	  // "PACKMLV2022".Admin.DisabledStatesCfg["LPMLV2022_MODE_INVALID"]     := "InstLPMLV2022_UnitModeStateManager".configuration.DisabledStatesCfg["LPMLV2022_MODE_INVALID"];
	  "PACKMLV2022".Admin.DisabledStatesCfg["LPMLV2022_MODE_PRODUCTION"]  := "InstLPMLV2022_UnitModeStateManager".configuration.DisabledStatesCfg["LPMLV2022_MODE_PRODUCTION"];
	  "PACKMLV2022".Admin.DisabledStatesCfg["LPMLV2022_MODE_MAINTENANCE"] := "InstLPMLV2022_UnitModeStateManager".configuration.DisabledStatesCfg["LPMLV2022_MODE_MAINTENANCE"];
	  "PACKMLV2022".Admin.DisabledStatesCfg["LPMLV2022_MODE_MANUAL"]      := "InstLPMLV2022_UnitModeStateManager".configuration.DisabledStatesCfg["LPMLV2022_MODE_MANUAL"];
	  "PACKMLV2022".Admin.DisabledStatesCfg["LPMLV2022_MODE_USER_01"]     := "InstLPMLV2022_UnitModeStateManager".configuration.DisabledStatesCfg["LPMLV2022_MODE_USER_01"];
	  // "PACKMLV2022".Admin.DisabledStatesCfg["LPMLV2022_MODE_USER_02"]     := "InstLPMLV2022_UnitModeStateManager".configuration.DisabledStatesCfg["LPMLV2022_MODE_USER_02"];
	  
	  "PACKMLV2022".Admin.CurDisabledStates := "InstLPMLV2022_UnitModeStateManager".CurDisabledStates;
	  
	  "PACKMLV2022".Admin.EnabledModesCfg := "InstLPMLV2022_UnitModeStateManager".configuration.EnabledModesCfg;
	  
	  // "PACKMLV2022".Admin.ModeTransitionCfg["LPMLV2022_MODE_INVALID"]     := "InstLPMLV2022_UnitModeStateManager".configuration.ModeTransitionCfg["LPMLV2022_MODE_INVALID"];
	  "PACKMLV2022".Admin.ModeTransitionCfg["LPMLV2022_MODE_PRODUCTION"]  := "InstLPMLV2022_UnitModeStateManager".configuration.ModeTransitionCfg["LPMLV2022_MODE_PRODUCTION"];
	  "PACKMLV2022".Admin.ModeTransitionCfg["LPMLV2022_MODE_MAINTENANCE"] := "InstLPMLV2022_UnitModeStateManager".configuration.ModeTransitionCfg["LPMLV2022_MODE_MAINTENANCE"];
	  "PACKMLV2022".Admin.ModeTransitionCfg["LPMLV2022_MODE_MANUAL"]      := "InstLPMLV2022_UnitModeStateManager".configuration.ModeTransitionCfg["LPMLV2022_MODE_MANUAL"];
	  "PACKMLV2022".Admin.ModeTransitionCfg["LPMLV2022_MODE_USER_01"]     := "InstLPMLV2022_UnitModeStateManager".configuration.ModeTransitionCfg["LPMLV2022_MODE_USER_01"];
	  // "PACKMLV2022".Admin.ModeTransitionCfg["LPMLV2022_MODE_USER_02"]     := "InstLPMLV2022_UnitModeStateManager".configuration.ModeTransitionCfg["LPMLV2022_MODE_USER_02"];
	  
	  // PLCDateTime
	  #tempReturnValue := RD_LOC_T(#tempPLCDateTimeDTL);
	  
	  "PACKMLV2022".Admin.PLCDateTime.Year        := UINT_TO_INT(#tempPLCDateTimeDTL.YEAR);
	  "PACKMLV2022".Admin.PLCDateTime.Month       := #tempPLCDateTimeDTL.MONTH;
	  "PACKMLV2022".Admin.PLCDateTime.Day         := #tempPLCDateTimeDTL.DAY;
	  "PACKMLV2022".Admin.PLCDateTime.Hour        := #tempPLCDateTimeDTL.HOUR;
	  "PACKMLV2022".Admin.PLCDateTime.Minute      := #tempPLCDateTimeDTL.MINUTE;
	  "PACKMLV2022".Admin.PLCDateTime.Second      := #tempPLCDateTimeDTL.SECOND;
	  "PACKMLV2022".Admin.PLCDateTime.Millisecond := UDINT_TO_INT(#tempPLCDateTimeDTL.NANOSECOND / 1000000);
	  
	  "PACKMLV2022".Admin.PLCDateTimeDTL := #tempPLCDateTimeDTL;
	END_REGION
END_FUNCTION_BLOCK

FUNCTION_BLOCK "LPMLV2022_UnitModeStateManagerBool"
TITLE = LPMLV2022_UnitModeStateManagerBool
{ S7_Optimized_Access := 'TRUE' }
AUTHOR : APC_ERLF
FAMILY : OMAC
VERSION : 1.0
//Support: tech.team.motioncontrol@siemens.com
   VAR_INPUT 
      ProductionModeRequest { S7_HiddenAssignment := 'Show'} : Bool;   // Rising edge: Request change to unit mode Production
      MaintenanceModeRequest { S7_HiddenAssignment := 'Show'} : Bool;   // Rising edge: Request change to unit mode Maintenance
      ManualModeRequest { S7_HiddenAssignment := 'Show'} : Bool;   // Rising edge: Request change to unit mode Manual
      UserMode01Request { S7_HiddenAssignment := 'Show'} : Bool;   // Rising edge: Request change to user-defined unit mode 01
      UserMode02Request : Bool;   // Rising edge: Request change to user-defined unit mode 02
      UserMode03Request : Bool;   // Rising edge: Request change to user-defined unit mode 03
      UserMode04Request : Bool;   // Rising edge: Request change to user-defined unit mode 04
      UserMode05Request : Bool;   // Rising edge: Request change to user-defined unit mode 05
      ResetCmdRequest { S7_HiddenAssignment := 'Show'} : Bool;   // Rising edge: Request control command Reset
      StartCmdRequest { S7_HiddenAssignment := 'Show'} : Bool;   // Rising edge: Request control command Start
      StopCmdRequest { S7_HiddenAssignment := 'Show'} : Bool;   // Rising edge: Request control command Stop
      HoldCmdRequest { S7_HiddenAssignment := 'Show'} : Bool;   // Rising edge: Request control command Hold
      UnholdCmdRequest { S7_HiddenAssignment := 'Show'} : Bool;   // Rising edge: Request control command Unhold
      SuspendCmdRequest { S7_HiddenAssignment := 'Show'} : Bool;   // Rising edge: Request control command Suspend
      UnsuspendCmdRequest { S7_HiddenAssignment := 'Show'} : Bool;   // Rising edge: Request control command Unsuspend
      AbortCmdRequest { S7_HiddenAssignment := 'Show'} : Bool;   // Rising edge: Request control command Abort
      ClearCmdRequest { S7_HiddenAssignment := 'Show'} : Bool;   // Rising edge: Request control command Clear
      CompleteCmdRequest { S7_HiddenAssignment := 'Show'} : Bool;   // Rising edge: Request control command Complete
      SC : Bool;   // State change from FALSE to TRUE (rising edge) triggers state complete signal
      configuration : "LPMLV2022_typeConfiguration" := ((), [()], [16#0, 31(16#0000_0214)], (), ());   // FB configuration (is taken into account in first call after STOP/RUN)
   END_VAR

   VAR_OUTPUT 
      UnitModeCurrent { ExternalWritable := 'False'} : DInt := "LPMLV2022_MODE_INVALID";   // Current unit mode
      StateCurrent { ExternalWritable := 'False'} : DInt := "LPMLV2022_STATE_UNDEFINED";   // Current state
      ProductionModeActive { ExternalWritable := 'False'; S7_HiddenAssignment := 'Show'} : Bool;   // TRUE: Unit mode Production is currently active
      MaintenanceModeActive { ExternalWritable := 'False'; S7_HiddenAssignment := 'Show'} : Bool;   // TRUE: Unit mode Maintenance is currently active
      ManualModeActive { ExternalWritable := 'False'; S7_HiddenAssignment := 'Show'} : Bool;   // TRUE: Unit mode Manual is currently active
      UserMode01Active { ExternalWritable := 'False'; S7_HiddenAssignment := 'Show'} : Bool;   // TRUE: User-defined unit mode 01 is currently active
      UserMode02Active { ExternalWritable := 'False'} : Bool;   // TRUE: User-defined unit mode 02 is currently active
      UserMode03Active { ExternalWritable := 'False'} : Bool;   // TRUE: User-defined unit mode 03 is currently active
      UserMode04Active { ExternalWritable := 'False'} : Bool;   // TRUE: User-defined unit mode 04 is currently active
      UserMode05Active { ExternalWritable := 'False'} : Bool;   // TRUE: User-defined unit mode 05 is currently active
      ClearingStateActive { ExternalWritable := 'False'; S7_HiddenAssignment := 'Show'} : Bool;   // TRUE: State Clearing is currently active
      StoppedStateActive { ExternalWritable := 'False'; S7_HiddenAssignment := 'Show'} : Bool;   // TRUE: State Stopped is currently active
      StartingStateActive { ExternalWritable := 'False'; S7_HiddenAssignment := 'Show'} : Bool;   // TRUE: State Starting is currently active
      IdleStateActive { ExternalWritable := 'False'; S7_HiddenAssignment := 'Show'} : Bool;   // TRUE: State Idle is currently active
      SuspendedStateActive { ExternalWritable := 'False'; S7_HiddenAssignment := 'Show'} : Bool;   // TRUE: State Suspended is currently active
      ExecuteStateActive { ExternalWritable := 'False'; S7_HiddenAssignment := 'Show'} : Bool;   // TRUE: State Execute is currently active
      StoppingStateActive { ExternalWritable := 'False'; S7_HiddenAssignment := 'Show'} : Bool;   // TRUE: State Stopping is currently active
      AbortingStateActive { ExternalWritable := 'False'; S7_HiddenAssignment := 'Show'} : Bool;   // TRUE: State Aborting is currently active
      AbortedStateActive { ExternalWritable := 'False'; S7_HiddenAssignment := 'Show'} : Bool;   // TRUE: State Aborted is currently active
      HoldingStateActive { ExternalWritable := 'False'; S7_HiddenAssignment := 'Show'} : Bool;   // TRUE: State Holding is currently active
      HeldStateActive { ExternalWritable := 'False'; S7_HiddenAssignment := 'Show'} : Bool;   // TRUE: State Held is currently active
      UnholdingStateActive { ExternalWritable := 'False'; S7_HiddenAssignment := 'Show'} : Bool;   // TRUE: State Unholding is currently active
      SuspendingStateActive { ExternalWritable := 'False'; S7_HiddenAssignment := 'Show'} : Bool;   // TRUE: State Suspending is currently active
      UnsuspendingStateActive { ExternalWritable := 'False'; S7_HiddenAssignment := 'Show'} : Bool;   // TRUE: State Unsuspending is currently active
      ResettingStateActive { ExternalWritable := 'False'; S7_HiddenAssignment := 'Show'} : Bool;   // TRUE: State Resetting is currently active
      CompletingStateActive { ExternalWritable := 'False'; S7_HiddenAssignment := 'Show'} : Bool;   // TRUE: State Completing is currently active
      CompletedStateActive { ExternalWritable := 'False'; S7_HiddenAssignment := 'Show'} : Bool;   // TRUE: State Completed is currently active
      unitModeChangeNotAllowed { ExternalWritable := 'False'} : Bool;   // TRUE: Requested unit mode change is not allowed (output is reset with the next successful unit mode change or if all corresponding request inputs are set to FALSE)
      cntrlCmdNotAllowed { ExternalWritable := 'False'} : Bool;   // TRUE: Control command is not allowed (output is reset with the next successful control command or if all corresponding request inputs are set to FALSE)
   END_VAR

   VAR 
      instUnitModeStateManager { ExternalWritable := 'False'; S7_SetPoint := 'False'} : "LPMLV2022_UnitModeStateManager";   // Instance of LPMLV2022_UnitModeStateManager
      statFirstCycle { ExternalAccessible := 'False'; ExternalVisible := 'False'; ExternalWritable := 'False'} : Bool := TRUE;   // First cycle of run
      statUnitModeCurrentInternalOld { ExternalAccessible := 'False'; ExternalVisible := 'False'; ExternalWritable := 'False'} : DInt := "LPMLV2022_MODE_INVALID";   // For edge detection
      statStateInternalOld { ExternalAccessible := 'False'; ExternalVisible := 'False'; ExternalWritable := 'False'} : DInt := "LPMLV2022_STATE_UNDEFINED";   // For edge detection
      statBooleanInterfaceModeOld { ExternalAccessible := 'False'; ExternalVisible := 'False'; ExternalWritable := 'False'} : DWord;   // For edge detection
      statBooleanInterfaceCmdOld { ExternalAccessible := 'False'; ExternalVisible := 'False'; ExternalWritable := 'False'} : Word;   // For edge detection
   END_VAR

   VAR_TEMP 
      tempBooleanInterfaceMode : DWord;   // Status of boolean Mode inputs
      tempBooleanInterfaceCmd : Word;   // Status of boolean Cmd inputs except abort and stop
   END_VAR


BEGIN
	REGION HEADER
	  //================================================================================
	  // SIEMENS AG
	  // (c)Copyright 2023 All Rights Reserved
	  //--------------------------------------------------------------------------------
	  // Library: LPMLV2022 
	  // Tested with: S7-1211 with FW version V4.2, S7-1511-1 PN with FW version V2.6
	  // Engineering: TIA Portal V15.1
	  // Restrictions: -
	  // Requirements: S7-1200 FW 4.2 / S7-1500 FW 2.6
	  // Functionality: Machine and Unit States according to ANSI/ISA-TR88.00.02-2022
	  //                (if the default settings are active at 'holdCmdCfg' and 'completeCmdCfg')
	  // Support: tech.team.motioncontrol@siemens.com
	  // Note: Parameter comments are only available in language 'English (United States)'
	  //--------------------------------------------------------------------------------
	  // Change log table:
	  // Version  Date        Expert in charge  Changes applied
	  // 01.00.00 28.02.2023  KT                First released version
	  //================================================================================
	END_REGION
	
	IF #statFirstCycle THEN // Initialize values in first cycle
	  #instUnitModeStateManager.configuration := #configuration; // Copy configuration from input
	  #statFirstCycle := FALSE;
	
	ELSE // As from second cycle
	  //--------------------------------------------------------------------------------------------------
	  // Evaluation of input parameters
	  //--------------------------------------------------------------------------------------------------
	  #instUnitModeStateManager.UnitModeChangeRequest := TRUE; // Change request static TRUE
	
	  // Collect unit mode from boolean inputs
	  #tempBooleanInterfaceMode.%X1  := #ProductionModeRequest;
	  #tempBooleanInterfaceMode.%X2  := #MaintenanceModeRequest;
	  #tempBooleanInterfaceMode.%X3  := #ManualModeRequest;
	  #tempBooleanInterfaceMode.%X4  := #UserMode01Request;
	  #tempBooleanInterfaceMode.%X5  := #UserMode02Request;
	  #tempBooleanInterfaceMode.%X6  := #UserMode03Request;
	  #tempBooleanInterfaceMode.%X7  := #UserMode04Request;
	  #tempBooleanInterfaceMode.%X8  := #UserMode05Request;
	// #tempBooleanInterfaceMode.%X9  := #UserMode06Request;
	// #tempBooleanInterfaceMode.%X10 := #UserMode07Request;
	// #tempBooleanInterfaceMode.%X11 := #UserMode08Request;
	// #tempBooleanInterfaceMode.%X12 := #UserMode09Request;
	// #tempBooleanInterfaceMode.%X13 := #UserMode10Request;
	// #tempBooleanInterfaceMode.%X14 := #UserMode11Request;
	// #tempBooleanInterfaceMode.%X15 := #UserMode12Request;
	// #tempBooleanInterfaceMode.%X16 := #UserMode13Request;
	// #tempBooleanInterfaceMode.%X17 := #UserMode14Request;
	// #tempBooleanInterfaceMode.%X18 := #UserMode15Request;
	// #tempBooleanInterfaceMode.%X19 := #UserMode16Request;
	// #tempBooleanInterfaceMode.%X20 := #UserMode17Request;
	// #tempBooleanInterfaceMode.%X21 := #UserMode18Request;
	// #tempBooleanInterfaceMode.%X22 := #UserMode19Request;
	// #tempBooleanInterfaceMode.%X23 := #UserMode20Request;
	// #tempBooleanInterfaceMode.%X24 := #UserMode21Request;
	// #tempBooleanInterfaceMode.%X25 := #UserMode22Request;
	// #tempBooleanInterfaceMode.%X26 := #UserMode23Request;
	// #tempBooleanInterfaceMode.%X27 := #UserMode24Request;
	// #tempBooleanInterfaceMode.%X28 := #UserMode25Request;
	// #tempBooleanInterfaceMode.%X29 := #UserMode26Request;
	// #tempBooleanInterfaceMode.%X30 := #UserMode27Request;
	// #tempBooleanInterfaceMode.%X31 := #UserMode28Request;
	    
	  // Selection indicator: Rising edge at input, Priority (in case of multiple selection): Manual, Maintenance, User Mode 01..28, Production
	  IF #tempBooleanInterfaceMode.%X3 AND NOT #statBooleanInterfaceModeOld.%X3 THEN
	    #instUnitModeStateManager.UnitMode := "LPMLV2022_MODE_MANUAL";
	  ELSIF #tempBooleanInterfaceMode.%X2 AND NOT #statBooleanInterfaceModeOld.%X2 THEN
	    #instUnitModeStateManager.UnitMode := "LPMLV2022_MODE_MAINTENANCE";
	  ELSIF #tempBooleanInterfaceMode.%X4 AND NOT #statBooleanInterfaceModeOld.%X4 THEN
	    #instUnitModeStateManager.UnitMode := "LPMLV2022_MODE_USER_01";
	  ELSIF #tempBooleanInterfaceMode.%X5 AND NOT #statBooleanInterfaceModeOld.%X5 THEN
	    #instUnitModeStateManager.UnitMode := "LPMLV2022_MODE_USER_02";
	  ELSIF #tempBooleanInterfaceMode.%X6 AND NOT #statBooleanInterfaceModeOld.%X6 THEN
	    #instUnitModeStateManager.UnitMode := "LPMLV2022_MODE_USER_03";
	  ELSIF #tempBooleanInterfaceMode.%X7 AND NOT #statBooleanInterfaceModeOld.%X7 THEN
	    #instUnitModeStateManager.UnitMode := "LPMLV2022_MODE_USER_04";
	  ELSIF #tempBooleanInterfaceMode.%X8 AND NOT #statBooleanInterfaceModeOld.%X8 THEN
	    #instUnitModeStateManager.UnitMode := "LPMLV2022_MODE_USER_05";
	// ELSIF #tempBooleanInterfaceMode.%X9 AND NOT #statBooleanInterfaceModeOld.%X9 THEN
	//   #instUnitModeStateManager.UnitMode := "LPMLV2022_MODE_USER_06";
	// ELSIF #tempBooleanInterfaceMode.%X10 AND NOT #statBooleanInterfaceModeOld.%X10 THEN
	//   #instUnitModeStateManager.UnitMode := "LPMLV2022_MODE_USER_07";
	// ELSIF #tempBooleanInterfaceMode.%X11 AND NOT #statBooleanInterfaceModeOld.%X11 THEN
	//   #instUnitModeStateManager.UnitMode := "LPMLV2022_MODE_USER_08";
	// ELSIF #tempBooleanInterfaceMode.%X12 AND NOT #statBooleanInterfaceModeOld.%X12 THEN
	//   #instUnitModeStateManager.UnitMode := "LPMLV2022_MODE_USER_09";
	// ELSIF #tempBooleanInterfaceMode.%X13 AND NOT #statBooleanInterfaceModeOld.%X13 THEN
	//   #instUnitModeStateManager.UnitMode := "LPMLV2022_MODE_USER_10";
	// ELSIF #tempBooleanInterfaceMode.%X14 AND NOT #statBooleanInterfaceModeOld.%X14 THEN
	//   #instUnitModeStateManager.UnitMode := "LPMLV2022_MODE_USER_11";
	// ELSIF #tempBooleanInterfaceMode.%X15 AND NOT #statBooleanInterfaceModeOld.%X15 THEN
	//   #instUnitModeStateManager.UnitMode := "LPMLV2022_MODE_USER_12";
	// ELSIF #tempBooleanInterfaceMode.%X16 AND NOT #statBooleanInterfaceModeOld.%X16 THEN
	//   #instUnitModeStateManager.UnitMode := "LPMLV2022_MODE_USER_13";
	// ELSIF #tempBooleanInterfaceMode.%X17 AND NOT #statBooleanInterfaceModeOld.%X17 THEN
	//   #instUnitModeStateManager.UnitMode := "LPMLV2022_MODE_USER_14";
	// ELSIF #tempBooleanInterfaceMode.%X18 AND NOT #statBooleanInterfaceModeOld.%X18 THEN
	//   #instUnitModeStateManager.UnitMode := "LPMLV2022_MODE_USER_15";
	// ELSIF #tempBooleanInterfaceMode.%X19 AND NOT #statBooleanInterfaceModeOld.%X19 THEN
	//   #instUnitModeStateManager.UnitMode := "LPMLV2022_MODE_USER_16";
	// ELSIF #tempBooleanInterfaceMode.%X20 AND NOT #statBooleanInterfaceModeOld.%X20 THEN
	//   #instUnitModeStateManager.UnitMode := "LPMLV2022_MODE_USER_17";
	// ELSIF #tempBooleanInterfaceMode.%X21 AND NOT #statBooleanInterfaceModeOld.%X21 THEN
	//   #instUnitModeStateManager.UnitMode := "LPMLV2022_MODE_USER_18";
	// ELSIF #tempBooleanInterfaceMode.%X22 AND NOT #statBooleanInterfaceModeOld.%X22 THEN
	//   #instUnitModeStateManager.UnitMode := "LPMLV2022_MODE_USER_19";
	// ELSIF #tempBooleanInterfaceMode.%X23 AND NOT #statBooleanInterfaceModeOld.%X23 THEN
	//   #instUnitModeStateManager.UnitMode := "LPMLV2022_MODE_USER_20";
	// ELSIF #tempBooleanInterfaceMode.%X24 AND NOT #statBooleanInterfaceModeOld.%X24 THEN
	//   #instUnitModeStateManager.UnitMode := "LPMLV2022_MODE_USER_21";
	// ELSIF #tempBooleanInterfaceMode.%X25 AND NOT #statBooleanInterfaceModeOld.%X25 THEN
	//   #instUnitModeStateManager.UnitMode := "LPMLV2022_MODE_USER_22";
	// ELSIF #tempBooleanInterfaceMode.%X26 AND NOT #statBooleanInterfaceModeOld.%X26 THEN
	//   #instUnitModeStateManager.UnitMode := "LPMLV2022_MODE_USER_23";
	// ELSIF #tempBooleanInterfaceMode.%X27 AND NOT #statBooleanInterfaceModeOld.%X27 THEN
	//   #instUnitModeStateManager.UnitMode := "LPMLV2022_MODE_USER_24";
	// ELSIF #tempBooleanInterfaceMode.%X28 AND NOT #statBooleanInterfaceModeOld.%X28 THEN
	//   #instUnitModeStateManager.UnitMode := "LPMLV2022_MODE_USER_25";
	// ELSIF #tempBooleanInterfaceMode.%X29 AND NOT #statBooleanInterfaceModeOld.%X29 THEN
	//   #instUnitModeStateManager.UnitMode := "LPMLV2022_MODE_USER_26";
	// ELSIF #tempBooleanInterfaceMode.%X30 AND NOT #statBooleanInterfaceModeOld.%X30 THEN
	//   #instUnitModeStateManager.UnitMode := "LPMLV2022_MODE_USER_27";
	// ELSIF #tempBooleanInterfaceMode.%X31 AND NOT #statBooleanInterfaceModeOld.%X31 THEN
	//   #instUnitModeStateManager.UnitMode := "LPMLV2022_MODE_USER_28";
	  ELSIF #tempBooleanInterfaceMode.%X1 AND NOT #statBooleanInterfaceModeOld.%X1 THEN
	    #instUnitModeStateManager.UnitMode := "LPMLV2022_MODE_PRODUCTION";
	  ELSIF #tempBooleanInterfaceMode = 16#0000_0000 THEN // all corresponding boolean request inputs are FALSE
	    #instUnitModeStateManager.UnitMode := "LPMLV2022_MODE_INVALID";
	  END_IF;
	  
	  #statBooleanInterfaceModeOld := #tempBooleanInterfaceMode; // Save values for edge detection
	  
	  // State complete signal
	  #instUnitModeStateManager.SC := #SC;
	  
	  // Evaluate CntrlCmd in boolean interface; priority descending: abort, stop, other commands
	  #instUnitModeStateManager.CmdChangeRequest := TRUE; // Change request static TRUE
	  
	  #tempBooleanInterfaceCmd.%X1 := #ResetCmdRequest;
	  #tempBooleanInterfaceCmd.%X2 := #StartCmdRequest;
	  #tempBooleanInterfaceCmd.%X3 := #StopCmdRequest;
	  #tempBooleanInterfaceCmd.%X4 := #HoldCmdRequest;
	  #tempBooleanInterfaceCmd.%X5 := #UnholdCmdRequest;
	  #tempBooleanInterfaceCmd.%X6 := #SuspendCmdRequest;
	  #tempBooleanInterfaceCmd.%X7 := #UnsuspendCmdRequest;
	  #tempBooleanInterfaceCmd.%X8 := #AbortCmdRequest;
	  #tempBooleanInterfaceCmd.%X9 := #ClearCmdRequest;
	  #tempBooleanInterfaceCmd.%X10 := #CompleteCmdRequest;
	  
	  // Selection indicator: Rising edge at input, Priority (in case of multiple selection): abort, stop, complete, reset, start, hold, unhold, suspend, unsuspend, clear
	  IF #tempBooleanInterfaceCmd.%X8 AND NOT #statBooleanInterfaceCmdOld.%X8 THEN
	    #instUnitModeStateManager.CntrlCmd := "LPMLV2022_CMD_ABORT";
	  ELSIF #tempBooleanInterfaceCmd.%X3 AND NOT #statBooleanInterfaceCmdOld.%X3 THEN
	    #instUnitModeStateManager.CntrlCmd := "LPMLV2022_CMD_STOP";
	  ELSIF #tempBooleanInterfaceCmd.%X10 AND NOT #statBooleanInterfaceCmdOld.%X10 THEN
	    #instUnitModeStateManager.CntrlCmd := "LPMLV2022_CMD_COMPLETE";
	  ELSIF #tempBooleanInterfaceCmd.%X1 AND NOT #statBooleanInterfaceCmdOld.%X1 THEN
	    #instUnitModeStateManager.CntrlCmd := "LPMLV2022_CMD_RESET";
	  ELSIF #tempBooleanInterfaceCmd.%X2 AND NOT #statBooleanInterfaceCmdOld.%X2 THEN
	    #instUnitModeStateManager.CntrlCmd := "LPMLV2022_CMD_START";
	  ELSIF #tempBooleanInterfaceCmd.%X4 AND NOT #statBooleanInterfaceCmdOld.%X4 THEN
	    #instUnitModeStateManager.CntrlCmd := "LPMLV2022_CMD_HOLD";
	  ELSIF #tempBooleanInterfaceCmd.%X5 AND NOT #statBooleanInterfaceCmdOld.%X5 THEN
	    #instUnitModeStateManager.CntrlCmd := "LPMLV2022_CMD_UNHOLD";
	  ELSIF #tempBooleanInterfaceCmd.%X6 AND NOT #statBooleanInterfaceCmdOld.%X6 THEN
	    #instUnitModeStateManager.CntrlCmd := "LPMLV2022_CMD_SUSPEND";
	  ELSIF #tempBooleanInterfaceCmd.%X7 AND NOT #statBooleanInterfaceCmdOld.%X7 THEN
	    #instUnitModeStateManager.CntrlCmd := "LPMLV2022_CMD_UNSUSPEND";
	  ELSIF #tempBooleanInterfaceCmd.%X9 AND NOT #statBooleanInterfaceCmdOld.%X9 THEN
	    #instUnitModeStateManager.CntrlCmd := "LPMLV2022_CMD_CLEAR";
	  ELSIF #tempBooleanInterfaceCmd = 16#0000_0000 THEN // all corresponding boolean request inputs are FALSE
	    #instUnitModeStateManager.CntrlCmd := "LPMLV2022_CMD_UNDEFINED";
	  END_IF;
	  
	  #statBooleanInterfaceCmdOld := #tempBooleanInterfaceCmd; // Save values for edge detection
	END_IF;
	
	//--------------------------------------------------------------------------------------------------
	// Call unit mode state manager
	//--------------------------------------------------------------------------------------------------
	#instUnitModeStateManager();
	
	//--------------------------------------------------------------------------------------------------
	// Write outputs including boolean interface outputs 
	//--------------------------------------------------------------------------------------------------
	#UnitModeCurrent := #instUnitModeStateManager.UnitModeCurrent;
	#StateCurrent    := #instUnitModeStateManager.StateCurrent;
	
	IF #instUnitModeStateManager.UnitModeCurrent <> #statUnitModeCurrentInternalOld THEN // Check if new unit mode is selected
	  #ProductionModeActive := FALSE;
	  #MaintenanceModeActive := FALSE;
	  #ManualModeActive := FALSE;
	  #UserMode01Active := FALSE;
	  #UserMode02Active := FALSE;
	  #UserMode03Active := FALSE;
	  #UserMode04Active := FALSE;
	  #UserMode05Active := FALSE;
	  // #UserMode06Active := FALSE;
	  // #UserMode07Active := FALSE;
	  // #UserMode08Active := FALSE;
	  // #UserMode09Active := FALSE;
	  // #UserMode10Active := FALSE;
	  // #UserMode11Active := FALSE;
	  // #UserMode12Active := FALSE;
	  // #UserMode13Active := FALSE;
	  // #UserMode14Active := FALSE;
	  // #UserMode15Active := FALSE;
	  // #UserMode16Active := FALSE;
	  // #UserMode17Active := FALSE;
	  // #UserMode18Active := FALSE;
	  // #UserMode19Active := FALSE;
	  // #UserMode20Active := FALSE;
	  // #UserMode21Active := FALSE;
	  // #UserMode22Active := FALSE;
	  // #UserMode23Active := FALSE;
	  // #UserMode24Active := FALSE;
	  // #UserMode25Active := FALSE;
	  // #UserMode26Active := FALSE;
	  // #UserMode27Active := FALSE;
	  // #UserMode28Active := FALSE;
	  
	  CASE #instUnitModeStateManager.UnitModeCurrent OF // Set new bit for current unit mode
	    "LPMLV2022_MODE_PRODUCTION":
	      #ProductionModeActive := TRUE;
	    "LPMLV2022_MODE_MAINTENANCE":
	      #MaintenanceModeActive := TRUE;
	    "LPMLV2022_MODE_MANUAL":
	      #ManualModeActive := TRUE;
	    "LPMLV2022_MODE_USER_01":
	      #UserMode01Active := TRUE;
	    "LPMLV2022_MODE_USER_02":
	      #UserMode02Active := TRUE;
	    "LPMLV2022_MODE_USER_03":
	      #UserMode03Active := TRUE;
	    "LPMLV2022_MODE_USER_04":
	      #UserMode04Active := TRUE;
	    "LPMLV2022_MODE_USER_05":
	      #UserMode05Active := TRUE;
	    // "LPMLV2022_MODE_USER_06":
	    //   #UserMode06Active := TRUE;
	    // "LPMLV2022_MODE_USER_07":
	    //   #UserMode07Active := TRUE;
	    // "LPMLV2022_MODE_USER_08":
	    //   #UserMode08Active := TRUE;
	    // "LPMLV2022_MODE_USER_09":
	    //   #UserMode09Active := TRUE;
	    // "LPMLV2022_MODE_USER_10":
	    //   #UserMode10Active := TRUE;
	    // "LPMLV2022_MODE_USER_11":
	    //   #UserMode11Active := TRUE;
	    // "LPMLV2022_MODE_USER_12":
	    //   #UserMode12Active := TRUE;
	    // "LPMLV2022_MODE_USER_13":
	    //   #UserMode13Active := TRUE;
	    // "LPMLV2022_MODE_USER_14":
	    //   #UserMode14Active := TRUE;
	    // "LPMLV2022_MODE_USER_15":
	    //   #UserMode15Active := TRUE;
	    // "LPMLV2022_MODE_USER_16":
	    //   #UserMode16Active := TRUE;
	    // "LPMLV2022_MODE_USER_17":
	    //   #UserMode17Active := TRUE;
	    // "LPMLV2022_MODE_USER_18":
	    //   #UserMode18Active := TRUE;
	    // "LPMLV2022_MODE_USER_19":
	    //   #UserMode19Active := TRUE;
	    // "LPMLV2022_MODE_USER_2"0:
	    //   #UserMode20Active := TRUE;
	    // "LPMLV2022_MODE_USER_21":
	    //   #UserMode21Active := TRUE;
	    // "LPMLV2022_MODE_USER_22":
	    //   #UserMode22Active := TRUE;
	    // "LPMLV2022_MODE_USER_23":
	    //   #UserMode23Active := TRUE;
	    // "LPMLV2022_MODE_USER_24":
	    //   #UserMode24Active := TRUE;
	    // "LPMLV2022_MODE_USER_25":
	    //   #UserMode25Active := TRUE;
	    // "LPMLV2022_MODE_USER_26":
	    //   #UserMode26Active := TRUE;
	    // "LPMLV2022_MODE_USER_27":
	    //   #UserMode27Active := TRUE;
	    // "LPMLV2022_MODE_USER_28":
	    //   #UserMode28Active := TRUE;
	    ELSE
	      ; // No bit is set
	  END_CASE;
	  
	  #statUnitModeCurrentInternalOld := #instUnitModeStateManager.UnitModeCurrent;
	END_IF;
	
	IF #instUnitModeStateManager.StateCurrent <> #statStateInternalOld THEN // Check if new state is selected 
	  // Set states of boolean interface outputs
	  // Delete old state
	  #ClearingStateActive := FALSE;
	  #StoppedStateActive := FALSE;
	  #StartingStateActive := FALSE;
	  #IdleStateActive := FALSE;
	  #SuspendedStateActive := FALSE;
	  #ExecuteStateActive := FALSE;
	  #StoppingStateActive := FALSE;
	  #AbortingStateActive := FALSE;
	  #AbortedStateActive := FALSE;
	  #HoldingStateActive := FALSE;
	  #HeldStateActive := FALSE;
	  #UnholdingStateActive := FALSE;
	  #SuspendingStateActive := FALSE;
	  #UnsuspendingStateActive := FALSE;
	  #ResettingStateActive := FALSE;
	  #CompletingStateActive := FALSE;
	  #CompletedStateActive := FALSE;
	  
	  // Set new state
	  CASE #instUnitModeStateManager.StateCurrent OF
	    "LPMLV2022_STATE_CLEARING":
	      #ClearingStateActive := TRUE;
	    "LPMLV2022_STATE_STOPPED":
	      #StoppedStateActive := TRUE;
	    "LPMLV2022_STATE_STARTING":
	      #StartingStateActive := TRUE;
	    "LPMLV2022_STATE_IDLE":
	      #IdleStateActive := TRUE;
	    "LPMLV2022_STATE_SUSPENDED":
	      #SuspendedStateActive := TRUE;
	    "LPMLV2022_STATE_EXECUTE":
	      #ExecuteStateActive := TRUE;
	    "LPMLV2022_STATE_STOPPING":
	      #StoppingStateActive := TRUE;
	    "LPMLV2022_STATE_ABORTING":
	      #AbortingStateActive := TRUE;
	    "LPMLV2022_STATE_ABORTED":
	      #AbortedStateActive := TRUE;
	    "LPMLV2022_STATE_HOLDING":
	      #HoldingStateActive := TRUE;
	    "LPMLV2022_STATE_HELD":
	      #HeldStateActive := TRUE;
	    "LPMLV2022_STATE_UNHOLDING":
	      #UnholdingStateActive := TRUE;
	    "LPMLV2022_STATE_SUSPENDING":
	      #SuspendingStateActive := TRUE;
	    "LPMLV2022_STATE_UNSUSPENDING":
	      #UnsuspendingStateActive := TRUE;
	    "LPMLV2022_STATE_RESETTING":
	      #ResettingStateActive := TRUE;
	    "LPMLV2022_STATE_COMPLETING":
	      #CompletingStateActive := TRUE;
	    "LPMLV2022_STATE_COMPLETED":
	      #CompletedStateActive := TRUE;
	    ELSE
	      ;
	  END_CASE; // End: Set new state
	  
	  #statStateInternalOld := #instUnitModeStateManager.StateCurrent;
	END_IF;// End: Write boolean interface outputs
	
	#unitModeChangeNotAllowed := #instUnitModeStateManager.unitModeChangeNotAllowed;
	#cntrlCmdNotAllowed       := #instUnitModeStateManager.cntrlCmdNotAllowed;
END_FUNCTION_BLOCK

FUNCTION "LPMLV2022_ConfigureCompleteCmdCfg" : Void
TITLE = LPMLV2022_ConfigureCompleteCmdCfg
{ S7_Optimized_Access := 'TRUE' }
AUTHOR : APC_ERLF
FAMILY : OMAC
VERSION : 1.0
//Support: tech.team.motioncontrol@siemens.com
   VAR_INPUT 
      Suspended : Bool;   // TRUE: The Complete control command is taken into account in state Suspended
      Execute : Bool;   // TRUE: The Complete control command is taken into account in state Execute
      Held : Bool;   // TRUE: The Complete control command is taken into account in state Held
   END_VAR

   VAR_OUTPUT 
      completeCmdCfg : DWord;   // Complete control command configuration for all unit modes (one config. for all modes). Bit locations within the DWORD value represent State numbers
   END_VAR


BEGIN
	REGION HEADER
	  //================================================================================
	  // SIEMENS AG
	  // (c)Copyright 2023 All Rights Reserved
	  //--------------------------------------------------------------------------------
	  // Library: LPMLV2022
	  // Tested with: S7-1211 with FW version V4.2, S7-1511-1 PN with FW version V2.6
	  // Engineering: TIA Portal V15.1
	  // Restrictions: -
	  // Requirements: S7-1200 FW 4.2 / S7-1500 FW 2.6
	  // Functionality: The function generates a DWord value which represents
	  //                the state configuration for all unit modes.
	  //                
	  //                Note: All inputs must be set to comply with ANSI/ISA-TR88.00.02-2022
	  //
	  // Support: tech.team.motioncontrol@siemens.com
	  // Note: Parameter comments are only available in language 'English (United States)'
	  //--------------------------------------------------------------------------------
	  // Change log table:
	  // Version  Date        Expert in charge  Changes applied
	  // 01.00.00 28.02.2023  KT                First released version
	  //================================================================================
	END_REGION
	
	// Initialize states configuration
	#completeCmdCfg := 16#0000_0000;
	
	// Set states configuration
	#completeCmdCfg.%X5  := #Suspended;
	#completeCmdCfg.%X6  := #Execute;
	#completeCmdCfg.%X11 := #Held;
END_FUNCTION

FUNCTION "LPMLV2022_ConfigureHoldCmdCfg" : Void
TITLE = LPMLV2022_ConfigureHoldCmdCfg
{ S7_Optimized_Access := 'TRUE' }
AUTHOR : APC_ERLF
FAMILY : OMAC
VERSION : 1.0
//Support: tech.team.motioncontrol@siemens.com
   VAR_INPUT 
      Starting : Bool;   // TRUE: The Hold control command is taken into account in state Starting
      Idle : Bool;   // TRUE: The Hold control command is taken into account in state Idle
      Suspended : Bool;   // TRUE: The Hold control command is taken into account in state Suspended
      Execute : Bool;   // TRUE: The Hold control command is taken into account in state Execute
      Unholding : Bool;   // TRUE: The Hold control command is taken into account in state Unholding
      Suspending : Bool;   // TRUE: The Hold control command is taken into account in state Suspending
      Unsuspending : Bool;   // TRUE: The Hold control command is taken into account in state Unsuspending
      Completing : Bool;   // TRUE: The Hold control command is taken into account in state Completing
      Completed : Bool;   // TRUE: The Hold control command is taken into account in state Completed
   END_VAR

   VAR_OUTPUT 
      holdCmdCfg : DWord;   // Hold control command configuration for all unit modes (one config. for all modes). Bit locations within the DWORD value represent State numbers
   END_VAR


BEGIN
	REGION HEADER
	  //================================================================================
	  // SIEMENS AG
	  // (c)Copyright 2023 All Rights Reserved
	  //--------------------------------------------------------------------------------
	  // Library: LPMLV2022
	  // Tested with: S7-1211 with FW version V4.2, S7-1511-1 PN with FW version V2.6
	  // Engineering: TIA Portal V15.1
	  // Restrictions: -
	  // Requirements: S7-1200 FW 4.2 / S7-1500 FW 2.6
	  // Functionality: The function generates a DWord value which represents
	  //                the state configuration for all unit modes.
	  //                
	  //                Note: Only the inputs 'Suspended' and 'Execute' must be set
	  //                      to comply with ANSI/ISA-TR88.00.02-2022
	  //                      
	  // Support: tech.team.motioncontrol@siemens.com
	  // Note: Parameter comments are only available in language 'English (United States)'
	  //--------------------------------------------------------------------------------
	  // Change log table:
	  // Version  Date        Expert in charge  Changes applied
	  // 01.00.00 28.02.2023  KT                First released version
	  //================================================================================
	END_REGION
	
	// Initialize states configuration
	#holdCmdCfg := 16#0000_0000;
	
	// Set states configuration
	#holdCmdCfg.%X3  := #Starting;
	#holdCmdCfg.%X4  := #Idle;
	#holdCmdCfg.%X5  := #Suspended;
	#holdCmdCfg.%X6  := #Execute;
	#holdCmdCfg.%X12 := #Unholding;
	#holdCmdCfg.%X13 := #Suspending;
	#holdCmdCfg.%X14 := #Unsuspending;
	#holdCmdCfg.%X16 := #Completing;
	#holdCmdCfg.%X17 := #Completed;
END_FUNCTION

FUNCTION "LPMLV2022_ConfigureModeTransitionCfg" : Void
TITLE = LPMLV2022_ConfigureModeTransitionCfg
{ S7_Optimized_Access := 'TRUE' }
AUTHOR : APC_ERLF
FAMILY : OMAC
VERSION : 1.0
//Support: tech.team.motioncontrol@siemens.com
   VAR_INPUT 
      Clearing : Bool;   // TRUE: Allow a mode transition to/from state Clearing
      Stopped : Bool;   // TRUE: Allow a mode transition to/from state Stopped
      Starting : Bool;   // TRUE: Allow a mode transition to/from state Starting
      Idle : Bool;   // TRUE: Allow a mode transition to/from state Idle
      Suspended : Bool;   // TRUE: Allow a mode transition to/from state Suspended
      Execute : Bool;   // TRUE: Allow a mode transition to/from state Execute
      Stopping : Bool;   // TRUE: Allow a mode transition to/from state Stopping
      Aborting : Bool;   // TRUE: Allow a mode transition to/from state Aborting
      Aborted : Bool;   // TRUE: Allow a mode transition to/from state Aborted
      Holding : Bool;   // TRUE: Allow a mode transition to/from state Holding
      Held : Bool;   // TRUE: Allow a mode transition to/from state Held
      Unholding : Bool;   // TRUE: Allow a mode transition to/from state Unholding
      Suspending : Bool;   // TRUE: Allow a mode transition to/from state Suspending
      Unsuspending : Bool;   // TRUE: Allow a mode transition to/from state Unsuspending
      Resetting : Bool;   // TRUE: Allow a mode transition to/from state Resetting
      Completing : Bool;   // TRUE: Allow a mode transition to/from state Completing
      Completed : Bool;   // TRUE: Allow a mode transition to/from state Completed
   END_VAR

   VAR_OUTPUT 
      ModeTransitionCfg : DWord;   // Mode Transition Configuration for one unit mode. Bit locations within the DWORD value represent State numbers
   END_VAR


BEGIN
	REGION HEADER
	  //================================================================================
	  // SIEMENS AG
	  // (c)Copyright 2023 All Rights Reserved
	  //--------------------------------------------------------------------------------
	  // Library: LPMLV2022
	  // Tested with: S7-1211 with FW version V4.2, S7-1511-1 PN with FW version V2.6
	  // Engineering: TIA Portal V15.1
	  // Restrictions: -
	  // Requirements: S7-1200 FW 4.2 / S7-1500 FW 2.6
	  // Functionality: The function generates a DWord value which represents
	  //                the state configuration for one unit mode.
	  // Support: tech.team.motioncontrol@siemens.com
	  // Note: Parameter comments are only available in language 'English (United States)'
	  //--------------------------------------------------------------------------------
	  // Change log table:
	  // Version  Date        Expert in charge  Changes applied
	  // 01.00.00 28.02.2023  KT                First released version
	  //================================================================================
	END_REGION
	
	// Initialize states configuration
	#ModeTransitionCfg := 16#0000_0000;
	
	// Set states configuration
	#ModeTransitionCfg.%X1  := #Clearing;
	#ModeTransitionCfg.%X2  := #Stopped;
	#ModeTransitionCfg.%X3  := #Starting;
	#ModeTransitionCfg.%X4  := #Idle;
	#ModeTransitionCfg.%X5  := #Suspended;
	#ModeTransitionCfg.%X6  := #Execute;
	#ModeTransitionCfg.%X7  := #Stopping;
	#ModeTransitionCfg.%X8  := #Aborting;
	#ModeTransitionCfg.%X9  := #Aborted;
	#ModeTransitionCfg.%X10 := #Holding;
	#ModeTransitionCfg.%X11 := #Held;
	#ModeTransitionCfg.%X12 := #Unholding;
	#ModeTransitionCfg.%X13 := #Suspending;
	#ModeTransitionCfg.%X14 := #Unsuspending;
	#ModeTransitionCfg.%X15 := #Resetting;
	#ModeTransitionCfg.%X16 := #Completing;
	#ModeTransitionCfg.%X17 := #Completed;
END_FUNCTION

FUNCTION_BLOCK "LPMLV2022_Stacklight"
TITLE = LPMLV2022_Stacklight
{ S7_Optimized_Access := 'TRUE' }
AUTHOR : APC_ERLF
FAMILY : OMAC
VERSION : 1.0
//Support: tech.team.motioncontrol@siemens.com
   VAR_INPUT 
      StateCurrent : DInt := "LPMLV2022_STATE_UNDEFINED";   // Current state
      starvedUpstream : Bool;   // TRUE: upstream system is not able to supply products
      blockedDownstream : Bool;   // TRUE: downstream system is not able to accept products
      materialLow : Bool;   // TRUE: low material
      materialExhausted : Bool;   // TRUE: material exhausted
   END_VAR

   VAR_OUTPUT 
      Stacklight { ExternalWritable := 'False'} : DWord;   // Indicator for the current stacklight status -> PackTags
      redSolid { ExternalWritable := 'False'} : Bool;   // Status of stacklight bit 0
      redFlashing { ExternalWritable := 'False'} : Bool;   // Status of stacklight bit 1
      amberSolid { ExternalWritable := 'False'} : Bool;   // Status of stacklight bit 2
      amberFlashing { ExternalWritable := 'False'} : Bool;   // Status of stacklight bit 3
      blueSolid { ExternalWritable := 'False'} : Bool;   // Status of stacklight bit 4
      blueFlashing { ExternalWritable := 'False'} : Bool;   // Status of stacklight bit 5
      greenSolid { ExternalWritable := 'False'} : Bool;   // Status of stacklight bit 6
      greenFlashing { ExternalWritable := 'False'} : Bool;   // Status of stacklight bit 7
      hornFlashing { ExternalWritable := 'False'} : Bool;   // Status of stacklight bit 9
   END_VAR

   VAR_TEMP 
      tempRedSolid : Bool;   // Status of stacklight bit 0
      tempRedFlashing : Bool;   // Status of stacklight bit 1
      tempAmberSolid : Bool;   // Status of stacklight bit 2
      tempAmberFlashing : Bool;   // Status of stacklight bit 3
      tempBlueSolid : Bool;   // Status of stacklight bit 4
      tempBlueFlashing : Bool;   // Status of stacklight bit 5
      tempGreenSolid : Bool;   // Status of stacklight bit 6
      tempGreenFlashing : Bool;   // Status of stacklight bit 7
      tempHornFlashing : Bool;   // Status of stacklight bit 9
   END_VAR


BEGIN
	REGION HEADER
	  //================================================================================
	  // SIEMENS AG
	  // (c)Copyright 2023 All Rights Reserved
	  //--------------------------------------------------------------------------------
	  // Library: LPMLV2022
	  // Tested with: S7-1211 with FW version V4.2, S7-1511-1 PN with FW version V2.6
	  // Engineering: TIA Portal V15.1
	  // Restrictions: -
	  // Requirements: S7-1200 FW 4.2 / S7-1500 FW 2.6
	  // Functionality: Stacklight status according to ANSI/ISA-TR88.00.02-2022
	  // Support: tech.team.motioncontrol@siemens.com
	  // Note: Parameter comments are only available in language 'English (United States)'
	  //--------------------------------------------------------------------------------
	  // Change log table:
	  // Version  Date        Expert in charge  Changes applied
	  // 01.00.00 28.02.2023  KT                First released version
	  //================================================================================
	END_REGION
	
	// Example of how the stacklight can be made to correspond to certain machine conditions and PackML States
	
	//                    |Aborting |Clearing | Aborted |Completed| Stopped |Stopping |Resetting|  Idle   |Starting |Execute  | Comple- | Holding |Held (No |Unholding| Suspen- |Suspended|Unsuspen-|                    
	//                    |         |         |         |         |         |         |         |         |         |         |  ting   |         |Product.)|         |  ding   |         |  ding   |                    
	//--------------------+---------+---------+---------+---------+---------+---------+---------+---------+---------+---------+---------+---------+---------+---------+---------+---------+---------+--------------------
	// Abnormal Stop      |    F    |    F    |    F    |         |         |         |         |         |         |         |         |         |         |         |         |         |         | Red Lamp Flashing  
	//--------------------+---------+---------+---------+---------+---------+---------+---------+---------+---------+---------+---------+---------+---------+---------+---------+---------+---------+--------------------
	// Controlled Stop    |         |         |         |    S    |    S    |    S    |    S    |         |         |         |         |         |         |         |         |         |         | Red Lamp Solid     
	//--------------------+---------+---------+---------+---------+---------+---------+---------+---------+---------+---------+---------+---------+---------+---------+---------+---------+---------+--------------------
	// Starved Upstream   |         |         |         |         |         |         |         |         |         |         |         |         |         |         |    F    |    F    |         | Amber Lamp Flashing
	//--------------------+---------+---------+---------+---------+---------+---------+---------+---------+---------+---------+---------+---------+---------+---------+---------+---------+---------+--------------------
	// Blocked Downstream |         |         |         |         |         |         |         |         |         |         |         |         |         |         |    S    |    S    |         | Amber Lamp Solid   
	//--------------------+---------+---------+---------+---------+---------+---------+---------+---------+---------+---------+---------+---------+---------+---------+---------+---------+---------+--------------------
	// Low Material       |    F    |    F    |    F    |    F    |    F    |    F    |    F    |    F    |    F    |    F    |    F    |         |         |    F    |    F    |    F    |    F    | Blue Lamp Flashing 
	//--------------------+---------+---------+---------+---------+---------+---------+---------+---------+---------+---------+---------+---------+---------+---------+---------+---------+---------+--------------------
	// Material Exhausted |         |         |         |         |         |         |         |         |         |         |         |    S    |    S    |         |         |         |         | Blue Lamp Solid    
	//--------------------+---------+---------+---------+---------+---------+---------+---------+---------+---------+---------+---------+---------+---------+---------+---------+---------+---------+--------------------
	// Ready to Start     |         |         |         |         |         |         |         |    F    |         |         |         |         |         |         |         |         |         | Green Lamp Flashing
	//--------------------+---------+---------+---------+---------+---------+---------+---------+---------+---------+---------+---------+---------+---------+---------+---------+---------+---------+--------------------
	// Running            |         |         |         |         |         |         |         |         |    S    |    S    |    S    |         |         |    S    |         |         |    S    | Green Lamp Solid   
	//--------------------+---------+---------+---------+---------+---------+---------+---------+---------+---------+---------+---------+---------+---------+---------+---------+---------+---------+--------------------
	// Starting/Restarting|         |         |         |         |         |         |         |         |    F    |         |         |         |         |    F    |         |         |    F    | Horn               
	//--------------------+---------+---------+---------+---------+---------+---------+---------+---------+---------+---------+---------+---------+---------+---------+---------+---------+---------+--------------------
	
	// The temporary variables are automatically set to FALSE, because the "Optimized block access" attribute is set
	
	CASE #StateCurrent OF
	  "LPMLV2022_STATE_EXECUTE":
	    #tempBlueFlashing := #materialLow;
	    #tempGreenSolid   := TRUE;
	    
	  "LPMLV2022_STATE_COMPLETING":
	    #tempBlueFlashing := #materialLow;
	    #tempGreenSolid   := TRUE;
	    
	  "LPMLV2022_STATE_COMPLETED":
	    #tempRedSolid     := TRUE;
	    #tempBlueFlashing := #materialLow;
	    
	  "LPMLV2022_STATE_RESETTING":
	    #tempRedSolid := TRUE;
	    #tempBlueFlashing := #materialLow;
	    
	  "LPMLV2022_STATE_IDLE":
	    #tempBlueFlashing  := #materialLow;
	    #tempGreenFlashing := TRUE;
	    
	  "LPMLV2022_STATE_STARTING":
	    #tempBlueFlashing := #materialLow;
	    #tempGreenSolid   := TRUE;
	    #tempHornFlashing := TRUE;
	    
	  "LPMLV2022_STATE_UNHOLDING":
	    #tempBlueFlashing := #materialLow;
	    #tempGreenSolid   := TRUE;
	    #tempHornFlashing := TRUE;
	    
	  "LPMLV2022_STATE_UNSUSPENDING":
	    #tempBlueFlashing := #materialLow;
	    #tempGreenSolid   := TRUE;
	    #tempHornFlashing := TRUE;
	    
	  "LPMLV2022_STATE_HOLDING":
	    #tempBlueSolid := #materialExhausted;
	    
	  "LPMLV2022_STATE_HELD":
	    #tempBlueSolid := #materialExhausted;
	    
	  "LPMLV2022_STATE_SUSPENDING":
	    #tempAmberFlashing := #starvedUpstream;
	    #tempAmberSolid    := #blockedDownstream;
	    #tempBlueFlashing  := #materialLow;
	    
	  "LPMLV2022_STATE_SUSPENDED":
	    #tempAmberFlashing := #starvedUpstream;
	    #tempAmberSolid    := #blockedDownstream;
	    #tempBlueFlashing  := #materialLow;
	    
	  "LPMLV2022_STATE_ABORTING":
	    #tempRedFlashing  := TRUE;
	    #tempBlueFlashing := #materialLow;
	    
	  "LPMLV2022_STATE_ABORTED":
	    #tempRedFlashing  := TRUE;
	    #tempBlueFlashing := #materialLow;
	    
	  "LPMLV2022_STATE_CLEARING":
	    #tempRedFlashing  := TRUE;
	    #tempBlueFlashing := #materialLow;
	    
	  "LPMLV2022_STATE_STOPPING":
	    #tempRedSolid     := TRUE;
	    #tempBlueFlashing := #materialLow;
	    
	  "LPMLV2022_STATE_STOPPED":
	    #tempRedSolid     := TRUE;
	    #tempBlueFlashing := #materialLow;
	
	  // ELSE 
	  //   ; // Reset all outputs
	END_CASE;
	
	// Write outputs
	#Stacklight := 16#0000_0000;
	
	#Stacklight.%X0 := #redSolid      := #tempRedSolid;
	#Stacklight.%X1 := #redFlashing   := #tempRedFlashing;
	#Stacklight.%X2 := #amberSolid    := #tempAmberSolid;
	#Stacklight.%X3 := #amberFlashing := #tempAmberFlashing;
	#Stacklight.%X4 := #blueSolid     := #tempBlueSolid;
	#Stacklight.%X5 := #blueFlashing  := #tempBlueFlashing;
	#Stacklight.%X6 := #greenSolid    := #tempGreenSolid;
	#Stacklight.%X7 := #greenFlashing := #tempGreenFlashing;
	#Stacklight.%X9 := #hornFlashing  := #tempHornFlashing;
END_FUNCTION_BLOCK

FUNCTION_BLOCK "LPMLV2022_UnitModeStateTimes"
TITLE = LPMLV2022_UnitModeStateTimes
{ S7_Optimized_Access := 'TRUE' }
AUTHOR : APC_ERLF
FAMILY : OMAC
VERSION : 1.0
//Support: tech.team.motioncontrol@siemens.com
   VAR_INPUT 
      UnitModeCurrent : DInt := "LPMLV2022_MODE_INVALID";   // Current unit mode
      StateCurrent : DInt := "LPMLV2022_STATE_UNDEFINED";   // Current state
      resetTimes : Bool;   // State change from FALSE to TRUE (rising edge) resets unit mode/state times and cumulative times
   END_VAR

   VAR_OUTPUT 
      ModeTimeCurrent { ExternalWritable := 'False'} : DInt;   // Actual time for current mode in seconds
      StateTimeCurrent { ExternalWritable := 'False'} : DInt;   // Actual time for current state in seconds
   END_VAR
   VAR_OUTPUT RETAIN
      AccTimeSinceReset { ExternalWritable := 'False'} : DInt;   // Accumulated time since last reset in seconds
   END_VAR
   VAR_OUTPUT 
      actualTimeAllModes { ExternalWritable := 'False'} : Array[0.."LPMLV2022_MODES_UPPER_LIM"] of DInt;   // Actual time for all modes in seconds (former name: ModeCurrentTime)
   END_VAR
   VAR_OUTPUT RETAIN
      cumulativeTimeAllModes { ExternalWritable := 'False'} : Array[0.."LPMLV2022_MODES_UPPER_LIM"] of DInt;   // Cumulative time for all modes in seconds (former name: ModeCumulativeTime)
   END_VAR
   VAR_OUTPUT 
      actualTimeAllStatesOfAllModes { ExternalWritable := 'False'} : Array[0.."LPMLV2022_MODES_UPPER_LIM", 0.."LPMLV2022_STATES_UPPER_LIM"] of DInt;   // Actual time for all states in seconds (former name: StateCurrentTime)
   END_VAR
   VAR_OUTPUT RETAIN
      cumulativeTimeAllStatesOfAllModes { ExternalWritable := 'False'} : Array[0.."LPMLV2022_MODES_UPPER_LIM", 0.."LPMLV2022_STATES_UPPER_LIM"] of DInt;   // Cumulative time for all states in seconds (former name: StateCumulativeTime)
   END_VAR
   VAR_OUTPUT 
      actualTimeAllStatesOfCurrentMode { ExternalWritable := 'False'} : Array[0.."LPMLV2022_STATES_UPPER_LIM"] of DInt;   // Actual time for all states in current mode in seconds
      cumulativeTimeAllStatesOfCurrentMode { ExternalWritable := 'False'} : Array[0.."LPMLV2022_STATES_UPPER_LIM"] of DInt;   // Cumulative time for all states in current mode in seconds
      cumulativeTimeCurrentMode { ExternalWritable := 'False'} : DInt;   // Cumulative time for current mode in seconds
   END_VAR

   VAR 
      statUnitModeCurrentOld { ExternalAccessible := 'False'; ExternalVisible := 'False'; ExternalWritable := 'False'} : DInt := "LPMLV2022_MODE_INVALID";   // For edge detection
      statStateCurrentOld { ExternalAccessible := 'False'; ExternalVisible := 'False'; ExternalWritable := 'False'} : DInt := "LPMLV2022_STATE_UNDEFINED";   // For edge detection
      statResetTimesOld { ExternalAccessible := 'False'; ExternalVisible := 'False'; ExternalWritable := 'False'} : Bool;   // For edge detection
      statStartingPointMeasureRuntime { ExternalAccessible := 'False'; ExternalVisible := 'False'; ExternalWritable := 'False'} : LReal;   // Saved value of runtime system function
      statRuntime { ExternalAccessible := 'False'; ExternalVisible := 'False'; ExternalWritable := 'False'} : LReal;   // Runtime variable
      statFirstCycle { ExternalAccessible := 'False'; ExternalVisible := 'False'; ExternalWritable := 'False'} : Bool := TRUE;   // First cycle of run
      statCurrentModeCurrentTime { ExternalAccessible := 'False'; ExternalVisible := 'False'; ExternalWritable := 'False'} : DInt;   // Actual time for current mode in seconds
      statCurrentStateCurrentTime { ExternalAccessible := 'False'; ExternalVisible := 'False'; ExternalWritable := 'False'} : DInt;   // Actual time for current state in seconds
   END_VAR

   VAR_TEMP 
      tempI : Int;   // Loop counter
      tempJ : Int;   // Loop counter
      tempMeasuredRuntime : LReal;   // Return value of RUNTIME instruction
      tempRuntimeIntegerPart : DInt;   // Runtime variable (integer part)
      tempUnitModeCurrent : DInt;   // Verified input value
      tempStateCurrent : DInt;   // Verified input value
   END_VAR


BEGIN
	REGION HEADER
	  //================================================================================
	  // SIEMENS AG
	  // (c)Copyright 2023 All Rights Reserved
	  //--------------------------------------------------------------------------------
	  // Library: LPMLV2022 
	  // Tested with: S7-1211 with FW version V4.2, S7-1511-1 PN with FW version V2.6
	  // Engineering: TIA Portal V15.1
	  // Restrictions: -
	  // Requirements: S7-1200 FW 4.2 / S7-1500 FW 2.6
	  // Functionality: Determination of unit modes and states times (current and also
	  //                cumulative times)
	  // Support: tech.team.motioncontrol@siemens.com
	  // Note: Parameter comments are only available in language 'English (United States)'
	  //--------------------------------------------------------------------------------
	  // Change log table:
	  // Version  Date        Expert in charge  Changes applied
	  // 01.00.00 28.02.2023  KT                First released version
	  //================================================================================
	END_REGION
	
	IF #statFirstCycle OR (#resetTimes AND NOT #statResetTimesOld) THEN
	  // Reset times structures
	  #statCurrentModeCurrentTime  := 0;
	  #statCurrentStateCurrentTime := 0;
	
	  FOR #tempI := "LPMLV2022_MODE_INVALID" TO "LPMLV2022_MODES_UPPER_LIM" DO
	    #actualTimeAllModes[#tempI] := 0;
	    IF NOT #statFirstCycle THEN // Do only with rising edge at resetTimes
	      #cumulativeTimeAllModes[#tempI] := 0;
	    END_IF;
	
	    FOR #tempJ := "LPMLV2022_STATE_UNDEFINED" TO "LPMLV2022_STATES_UPPER_LIM" DO
	      #actualTimeAllStatesOfAllModes[#tempI, #tempJ] := 0;
	      IF NOT #statFirstCycle THEN // Do only with rising edge at resetTimes
	        #cumulativeTimeAllStatesOfAllModes[#tempI, #tempJ] := 0;
	      END_IF;
	    END_FOR;
	  END_FOR;
	
	  IF NOT #statFirstCycle THEN // Do only with rising edge at resetTimes
	    #AccTimeSinceReset := 0;
	  END_IF;
	  
	  // Reset additional outputs
	  #ModeTimeCurrent  := 0;
	  #StateTimeCurrent := 0;
	
	  IF NOT #statFirstCycle THEN // Do only with rising edge at resetTimes
	    #cumulativeTimeCurrentMode := 0;
	  END_IF;
	
	  FOR #tempI := "LPMLV2022_STATE_UNDEFINED" TO "LPMLV2022_STATES_UPPER_LIM" DO
	    #actualTimeAllStatesOfCurrentMode[#tempI] := 0;
	    IF NOT #statFirstCycle THEN // Do only with rising edge at resetTimes
	      #cumulativeTimeAllStatesOfCurrentMode[#tempI] := 0;
	    END_IF;
	  END_FOR;
	
	  // Set starting point for calculation of elapsed seconds
	  #tempMeasuredRuntime := RUNTIME(#statStartingPointMeasureRuntime);
	  #statRuntime := 0.0;
	  
	  IF #statFirstCycle THEN
	    #statFirstCycle := FALSE;
	    RETURN; // Nothing else in this cycle to avoid runtime peaks
	  END_IF;
	END_IF;
	
	// Inputs UnitModeCurrent and StateCurrent
	#tempUnitModeCurrent := #UnitModeCurrent;
	#tempStateCurrent    := #StateCurrent;
	
	// Measure program runtime
	#tempMeasuredRuntime := RUNTIME(#statStartingPointMeasureRuntime);
	IF #tempMeasuredRuntime > 0.0 THEN // Value OK
	  #statRuntime := #statRuntime + #tempMeasuredRuntime;
	END_IF;
	
	// Check if at least one second has been reached
	IF #statRuntime > 1.0 THEN
	  #tempRuntimeIntegerPart := TRUNC_DINT(#statRuntime);
	  
	  IF #statUnitModeCurrentOld >= "LPMLV2022_MODE_INVALID" AND #statUnitModeCurrentOld <= "LPMLV2022_MODES_UPPER_LIM" THEN
	    // DINT overflow is not taken into account, because DINT in seconds means approx. 68 years
	    //#ModeCurrentTime[#statUnitModeCurrentOld] := #ModeCurrentTime[#statUnitModeCurrentOld] + #tempRuntimeIntegerPart;
	    #statCurrentModeCurrentTime := #statCurrentModeCurrentTime + #tempRuntimeIntegerPart;
	    #actualTimeAllModes[#statUnitModeCurrentOld] := #statCurrentModeCurrentTime;
	    #cumulativeTimeAllModes[#statUnitModeCurrentOld] := #cumulativeTimeAllModes[#statUnitModeCurrentOld] + #tempRuntimeIntegerPart;
	    
	    IF #statStateCurrentOld >= "LPMLV2022_STATE_UNDEFINED" AND #statStateCurrentOld <= "LPMLV2022_STATES_UPPER_LIM" THEN
	      // DINT overflow is not taken into account, because DINT in seconds means approx. 68 years
	      #statCurrentStateCurrentTime := #statCurrentStateCurrentTime + #tempRuntimeIntegerPart;
	      #actualTimeAllStatesOfAllModes[#statUnitModeCurrentOld, #statStateCurrentOld] := #statCurrentStateCurrentTime;
	      #cumulativeTimeAllStatesOfAllModes[#statUnitModeCurrentOld, #statStateCurrentOld] := #cumulativeTimeAllStatesOfAllModes[#statUnitModeCurrentOld, #statStateCurrentOld] + #tempRuntimeIntegerPart;
	    END_IF;
	  END_IF;
	
	  // DINT overflow is not taken into account, because DINT in seconds means approx. 68 years
	  #AccTimeSinceReset := #AccTimeSinceReset + #tempRuntimeIntegerPart;
	
	  #statRuntime := #statRuntime - #tempRuntimeIntegerPart; // Fractional part of runtime variable for next cycle
	END_IF;
	
	// Check if new unitMode is selected
	IF #tempUnitModeCurrent <> #statUnitModeCurrentOld THEN
	  IF #tempUnitModeCurrent >= "LPMLV2022_MODE_INVALID" AND #tempUnitModeCurrent <= "LPMLV2022_MODES_UPPER_LIM" THEN
	    #statCurrentModeCurrentTime := 0;
	    #actualTimeAllModes[#tempUnitModeCurrent] := 0;
	    IF #tempStateCurrent >= "LPMLV2022_STATE_UNDEFINED" AND #tempStateCurrent <= "LPMLV2022_STATES_UPPER_LIM" THEN
	      #statCurrentStateCurrentTime := 0;
	      #actualTimeAllStatesOfAllModes[#tempUnitModeCurrent, #tempStateCurrent] := 0;
	    END_IF;
	  END_IF;
	  
	  // Check if new state is selected  
	ELSIF #tempStateCurrent <> #statStateCurrentOld THEN
	  IF #tempUnitModeCurrent >= "LPMLV2022_MODE_INVALID" AND #tempUnitModeCurrent <= "LPMLV2022_MODES_UPPER_LIM" AND
	    #tempStateCurrent >= "LPMLV2022_STATE_UNDEFINED" AND #tempStateCurrent <= "LPMLV2022_STATES_UPPER_LIM"
	  THEN
	    #statCurrentStateCurrentTime := 0;
	    #actualTimeAllStatesOfAllModes[#tempUnitModeCurrent, #tempStateCurrent] := 0;
	  END_IF;
	END_IF;
	
	// Update additional outputs
	IF #tempUnitModeCurrent >= "LPMLV2022_MODE_INVALID" AND #tempUnitModeCurrent <= "LPMLV2022_MODES_UPPER_LIM" THEN
	  #ModeTimeCurrent           := #statCurrentModeCurrentTime;
	  #cumulativeTimeCurrentMode := #cumulativeTimeAllModes[#tempUnitModeCurrent];
	
	  IF #tempStateCurrent >= "LPMLV2022_STATE_UNDEFINED" AND #tempStateCurrent <= "LPMLV2022_STATES_UPPER_LIM" THEN
	    #StateTimeCurrent := #statCurrentStateCurrentTime;
	    #actualTimeAllStatesOfCurrentMode := #actualTimeAllStatesOfAllModes[#tempUnitModeCurrent];
	    #cumulativeTimeAllStatesOfCurrentMode := #cumulativeTimeAllStatesOfAllModes[#tempUnitModeCurrent];
	  ELSE
	    #StateTimeCurrent := 0;
	
	    FOR #tempI := "LPMLV2022_STATE_UNDEFINED" TO "LPMLV2022_STATES_UPPER_LIM" DO
	      #actualTimeAllStatesOfCurrentMode[#tempI]     := 0;
	      #cumulativeTimeAllStatesOfCurrentMode[#tempI] := 0;
	    END_FOR;
	  END_IF;
	
	ELSE
	  #ModeTimeCurrent  := 0;
	  #StateTimeCurrent := 0;
	  #cumulativeTimeCurrentMode := 0;
	  
	  FOR #tempI := "LPMLV2022_STATE_UNDEFINED" TO "LPMLV2022_STATES_UPPER_LIM" DO
	    #actualTimeAllStatesOfCurrentMode[#tempI]     := 0;
	    #cumulativeTimeAllStatesOfCurrentMode[#tempI] := 0;
	  END_FOR;
	END_IF;
	
	// Save values for state change detection
	#statUnitModeCurrentOld := #tempUnitModeCurrent;
	#statStateCurrentOld    := #tempStateCurrent;
	#statResetTimesOld := #resetTimes;
END_FUNCTION_BLOCK

DATA_BLOCK "PACKMLV2022"   // DB30135
TITLE = PackTags DB
{ S7_Optimized_Access := 'TRUE' }
VERSION : 0.1
// stored: AutoNumber true, DBAccessibleFromOPCUA true, DBAccessibleFromWebserver true, InstanceOfName LPMLV2022_typePackTags, InstanceOfType UDT, IsOnlyStoredInLoadMemory false, IsWriteProtectedInAS false
"LPMLV2022_typePackTags"
BEGIN
END_DATA_BLOCK

DATA_BLOCK "InstCallUnitModeStateManager"   // DB30130
{ DB_Accessible_From_OPC_UA := 'FALSE' }
VERSION : 0.1
// stored: AutoNumber true, DBAccessibleFromOPCUA false, DBAccessibleFromWebserver false, InstanceOfName CallUnitModeStateManager, InstanceOfType FB
"CallUnitModeStateManager"
BEGIN
END_DATA_BLOCK

DATA_BLOCK "InstLPMLV2022_Stacklight"   // DB30113
{ DB_Accessible_From_OPC_UA := 'FALSE' }
AUTHOR : APC_ERLF
FAMILY : OMAC
VERSION : 1.0
// stored: AutoNumber true, DBAccessibleFromOPCUA false, DBAccessibleFromWebserver false, InstanceOfName LPMLV2022_Stacklight, InstanceOfType FB
"LPMLV2022_Stacklight"
BEGIN
END_DATA_BLOCK

DATA_BLOCK "InstLPMLV2022_UnitModeStateManager"   // DB30110
{ DB_Accessible_From_OPC_UA := 'FALSE' }
AUTHOR : APC_ERLF
FAMILY : OMAC
VERSION : 1.0
// stored: AutoNumber true, DBAccessibleFromOPCUA false, DBAccessibleFromWebserver false, InstanceOfName LPMLV2022_UnitModeStateManager, InstanceOfType FB
"LPMLV2022_UnitModeStateManager"
   // VAR_INPUT
   //    UnitMode : DInt;
   //    UnitModeChangeRequest : Bool;
   //    CntrlCmd : DInt;
   //    CmdChangeRequest : Bool;
   //    SC : Bool;
   //    configuration : "LPMLV2022_typeConfiguration";
   // END_VAR
   // VAR_OUTPUT
   //    UnitModeCurrent { ExternalWritable := 'False'} : DInt;
   //    StateCurrent { ExternalWritable := 'False'} : DInt;
   //    StateRequested { ExternalWritable := 'False'} : DInt;
   //    StateChangeInProcess { ExternalWritable := 'False'} : Bool;
   //    CurDisabledStates { ExternalWritable := 'False'} : DWord;
   //    curHoldCmdCfg { ExternalWritable := 'False'} : DWord;
   //    curCompleteCmdCfg { ExternalWritable := 'False'} : DWord;
   //    unitModeChangeNotAllowed { ExternalWritable := 'False'} : Bool;
   //    cntrlCmdNotAllowed { ExternalWritable := 'False'} : Bool;
   //    diagnostics { ExternalWritable := 'False'} : "LPMLV2022_typeDiagnostics";
   // END_VAR
   // VAR
   //    statConfiguration { ExternalAccessible := 'False'; ExternalVisible := 'False'; ExternalWritable := 'False'} : "LPMLV2022_typeConfiguration";
   //    statUnitModeChangeRequest { ExternalAccessible := 'False'; ExternalVisible := 'False'; ExternalWritable := 'False'} : Bool;
   //    statCmdChangeRequest { ExternalAccessible := 'False'; ExternalVisible := 'False'; ExternalWritable := 'False'} : Bool;
   //    statFirstCycle { ExternalAccessible := 'False'; ExternalVisible := 'False'; ExternalWritable := 'False'} : Bool;
   //    statSCOld { ExternalAccessible := 'False'; ExternalVisible := 'False'; ExternalWritable := 'False'} : Bool;
   //    statUnitMode { ExternalAccessible := 'False'; ExternalVisible := 'False'; ExternalWritable := 'False'} : DInt;
   //    statUnitModeOld { ExternalAccessible := 'False'; ExternalVisible := 'False'; ExternalWritable := 'False'} : DInt;
   //    statUnitModeCurrentInternal { ExternalAccessible := 'False'; ExternalVisible := 'False'; ExternalWritable := 'False'} : DInt;
   //    statUnitModeCurrentInternalOld { ExternalAccessible := 'False'; ExternalVisible := 'False'; ExternalWritable := 'False'} : DInt;
   //    statStateCurrentOld { ExternalAccessible := 'False'; ExternalVisible := 'False'; ExternalWritable := 'False'} : DInt;
   //    statStateInternal { ExternalAccessible := 'False'; ExternalVisible := 'False'; ExternalWritable := 'False'} : DInt;
   //    statStateInternalOld { ExternalAccessible := 'False'; ExternalVisible := 'False'; ExternalWritable := 'False'} : DInt;
   //    statCntrlCmdOld { ExternalAccessible := 'False'; ExternalVisible := 'False'; ExternalWritable := 'False'} : DInt;
   //    statStatesInCurrentMode { ExternalAccessible := 'False'; ExternalVisible := 'False'; ExternalWritable := 'False'} : Struct
   //       clearing { ExternalAccessible := 'False'; ExternalVisible := 'False'; ExternalWritable := 'False'} : Bool;
   //       stopped { ExternalAccessible := 'False'; ExternalVisible := 'False'; ExternalWritable := 'False'} : Bool;
   //       starting { ExternalAccessible := 'False'; ExternalVisible := 'False'; ExternalWritable := 'False'} : Bool;
   //       idle { ExternalAccessible := 'False'; ExternalVisible := 'False'; ExternalWritable := 'False'} : Bool;
   //       suspended { ExternalAccessible := 'False'; ExternalVisible := 'False'; ExternalWritable := 'False'} : Bool;
   //       execute { ExternalAccessible := 'False'; ExternalVisible := 'False'; ExternalWritable := 'False'} : Bool;
   //       stopping { ExternalAccessible := 'False'; ExternalVisible := 'False'; ExternalWritable := 'False'} : Bool;
   //       aborting { ExternalAccessible := 'False'; ExternalVisible := 'False'; ExternalWritable := 'False'} : Bool;
   //       aborted { ExternalAccessible := 'False'; ExternalVisible := 'False'; ExternalWritable := 'False'} : Bool;
   //       holding { ExternalAccessible := 'False'; ExternalVisible := 'False'; ExternalWritable := 'False'} : Bool;
   //       held { ExternalAccessible := 'False'; ExternalVisible := 'False'; ExternalWritable := 'False'} : Bool;
   //       unholding { ExternalAccessible := 'False'; ExternalVisible := 'False'; ExternalWritable := 'False'} : Bool;
   //       suspending { ExternalAccessible := 'False'; ExternalVisible := 'False'; ExternalWritable := 'False'} : Bool;
   //       unsuspending { ExternalAccessible := 'False'; ExternalVisible := 'False'; ExternalWritable := 'False'} : Bool;
   //       resetting { ExternalAccessible := 'False'; ExternalVisible := 'False'; ExternalWritable := 'False'} : Bool;
   //       completing { ExternalAccessible := 'False'; ExternalVisible := 'False'; ExternalWritable := 'False'} : Bool;
   //       completed { ExternalAccessible := 'False'; ExternalVisible := 'False'; ExternalWritable := 'False'} : Bool;
   //    END_STRUCT;
   //    statConsiderHoldCmdIn { ExternalAccessible := 'False'; ExternalVisible := 'False'; ExternalWritable := 'False'} : Struct
   //       starting { ExternalAccessible := 'False'; ExternalVisible := 'False'; ExternalWritable := 'False'} : Bool;
   //       idle { ExternalAccessible := 'False'; ExternalVisible := 'False'; ExternalWritable := 'False'} : Bool;
   //       suspended { ExternalAccessible := 'False'; ExternalVisible := 'False'; ExternalWritable := 'False'} : Bool;
   //       execute { ExternalAccessible := 'False'; ExternalVisible := 'False'; ExternalWritable := 'False'} : Bool;
   //       unholding { ExternalAccessible := 'False'; ExternalVisible := 'False'; ExternalWritable := 'False'} : Bool;
   //       suspending { ExternalAccessible := 'False'; ExternalVisible := 'False'; ExternalWritable := 'False'} : Bool;
   //       unsuspending { ExternalAccessible := 'False'; ExternalVisible := 'False'; ExternalWritable := 'False'} : Bool;
   //       completing { ExternalAccessible := 'False'; ExternalVisible := 'False'; ExternalWritable := 'False'} : Bool;
   //       completed { ExternalAccessible := 'False'; ExternalVisible := 'False'; ExternalWritable := 'False'} : Bool;
   //    END_STRUCT;
   //    statConsiderCompleteCmdIn { ExternalAccessible := 'False'; ExternalVisible := 'False'; ExternalWritable := 'False'} : Struct
   //       suspended { ExternalAccessible := 'False'; ExternalVisible := 'False'; ExternalWritable := 'False'} : Bool;
   //       execute { ExternalAccessible := 'False'; ExternalVisible := 'False'; ExternalWritable := 'False'} : Bool;
   //       held { ExternalAccessible := 'False'; ExternalVisible := 'False'; ExternalWritable := 'False'} : Bool;
   //    END_STRUCT;
   //    statCmdChangeRequestOld { ExternalAccessible := 'False'; ExternalVisible := 'False'; ExternalWritable := 'False'} : Bool;
   //    statUnitModeChangeRequestOld { ExternalAccessible := 'False'; ExternalVisible := 'False'; ExternalWritable := 'False'} : Bool;
   //    statDiagnosticsBufferIndex { ExternalAccessible := 'False'; ExternalVisible := 'False'; ExternalWritable := 'False'} : Int;
   //    statStateRequested { ExternalAccessible := 'False'; ExternalVisible := 'False'; ExternalWritable := 'False'} : DInt;
   //    statUnitModeChangeNotAllowed { ExternalAccessible := 'False'; ExternalVisible := 'False'; ExternalWritable := 'False'} : Bool;
   //    statCntrlCmdNotAllowed { ExternalAccessible := 'False'; ExternalVisible := 'False'; ExternalWritable := 'False'} : Bool;
   // END_VAR
BEGIN
END_DATA_BLOCK

DATA_BLOCK "InstLPMLV2022_UnitModeStateTimes"   // DB30112
{ DB_Accessible_From_OPC_UA := 'FALSE' }
AUTHOR : APC_ERLF
FAMILY : OMAC
VERSION : 1.0
// stored: AutoNumber true, DBAccessibleFromOPCUA false, DBAccessibleFromWebserver false, InstanceOfName LPMLV2022_UnitModeStateTimes, InstanceOfType FB
"LPMLV2022_UnitModeStateTimes"
BEGIN
END_DATA_BLOCK

DATA_BLOCK "InstPACKMLV2022_PackTagsGlueCode"   // DB30132
{ DB_Accessible_From_OPC_UA := 'FALSE' }
VERSION : 0.1
// stored: AutoNumber true, DBAccessibleFromOPCUA false, DBAccessibleFromWebserver false, InstanceOfName PACKMLV2022_PackTagsGlueCode, InstanceOfType FB
"PACKMLV2022_PackTagsGlueCode"
BEGIN
END_DATA_BLOCK

DATA_BLOCK "InstShowUnitModeStateManagerDiagnosticsInHMI"   // DB30131
{ DB_Accessible_From_OPC_UA := 'FALSE' }
VERSION : 0.1
// stored: AutoNumber true, DBAccessibleFromOPCUA false, DBAccessibleFromWebserver false, InstanceOfName ShowUnitModeStateManagerDiagnosticsInHMI, InstanceOfType FB
"ShowUnitModeStateManagerDiagnosticsInHMI"
BEGIN
END_DATA_BLOCK
